(* IEC 61131-3 sources: st-fmt/tests/fixtures/comments, 6 files *)

(* ---- block_comments.expected.st ---- *)
(* A multi-line header
   that must keep
   its own layout *)
FUNCTION_BLOCK FB_Block
VAR
    a : UINT;  (* trailing block *)
END_VAR

x := y;  (* inline *)
z := 1;

END_FUNCTION_BLOCK

(* ---- block_comments.st ---- *)
(* A multi-line header
   that must keep
   its own layout *)
FUNCTION_BLOCK FB_Block
VAR
a : UINT; (* trailing block *)
END_VAR
x := (* inline *) y;
z := 1;
END_FUNCTION_BLOCK

(* ---- placement.expected.st ---- *)
/// Doc comment on the POU
FUNCTION_BLOCK FB_Documented
VAR
    n : INT;  // trailing on a declaration
    // a note before END_VAR
END_VAR

// leading the body
n := 1;  // trailing a statement
IF n > 0 THEN
    // inside a branch
    n := 2;
    // before END_IF
END_IF

END_FUNCTION_BLOCK

(* ---- placement.st ---- *)
/// Doc comment on the POU
FUNCTION_BLOCK FB_Documented
VAR
n : INT; // trailing on a declaration
// a note before END_VAR
END_VAR
// leading the body
n := 1; // trailing a statement
IF n > 0 THEN
// inside a branch
n := 2;
// before END_IF
END_IF
END_FUNCTION_BLOCK

(* ---- regions.expected.st ---- *)
FUNCTION_BLOCK FB_Regions
VAR
    {attribute 'symbol' := 'readwrite'}
    /// If true the run is stopped
    StopOnError : BOOL;

    (* Public vars *)

    /// Current state
    {attribute 'symbol' := 'read'}
    State : TestState;
END_VAR

{region Event logic}
    above := value >= threshold;
{endregion}

END_FUNCTION_BLOCK

(* ---- regions.st ---- *)
FUNCTION_BLOCK FB_Regions
VAR
{attribute 'symbol' := 'readwrite'}
/// If true the run is stopped
StopOnError : BOOL;

(* Public vars *)

/// Current state
{attribute 'symbol' := 'read'}
State : TestState;
END_VAR
{region Event logic}
above := value >= threshold;
{endregion}
END_FUNCTION_BLOCK
